(* IEC 61131-3 sources: std_i2980_v2.06_cp053/Source/IMM/ieccontrol/ExceptionInterpretation1 (part 2) *)

(* ---- FBODCErrorHandler.pu ---- *)
IMPORT_OVER_LISTFILE
 tyAlarmParams
, tySubID

END_IMPORT

FUNCTION_BLOCK FBODCErrorHandler #DUMMY_EDIT_BLOCK

VAR_INPUT
 iErrorKind : INT;
 iComponentNr : DINT;
 iErrorNr : DINT;
 AlarmParameters : tyAlarmParams;
END_VAR

VAR_IN_OUT
 SubID : tySubID;
END_VAR

VAR_OUTPUT
 bOpenWatchdog : BOOL;
 bSetAlarm : BOOL;
 AlarmID : ALARM;
 sParam1 : STRING(255);
 sParam2 : STRING(255);
END_VAR

SYSTEM_OBJECT
 erODCBuilderGeneralError : ALARM;
 erODCBuilderNoSignature : ALARM;
 erODCBuilderFileformat : ALARM;
 erODCBuilderInvalidSignature : ALARM;
 erODCBuilderInsertPosNotAvail : ALARM;
 erODCBuilderInsertBefNotAllow : ALARM;
 erODCBuilderInsertAfterNotAllow : ALARM;
 erODCBuilderMoveNotAvailable : ALARM;
 erODCBuilderError : ALARM;
 erODCBuilderSyntaxError : ALARM;
 erODCBuilderWarning : ALARM;
 erODCBuilderWarningFile : ALARM;
 erODCBuilderMultipleBaseSequ : ALARM;
 erODCBuilderPriorityCollision : ALARM;
 erODCBuilderBaseSeqNotFound : ALARM;
 erODCBuilderInstancePriority : ALARM;
 erODCBuilderParserException : ALARM;
 erODCCouldNotCreateLogFile : ALARM;
 erODCBuilderFirstMovement : ALARM;
 erODCBuilderLastMovement : ALARM;
 erODCBuilderSelectorVarValue : ALARM;
 erODCBuilderIllegalDominantMove : ALARM;
 erODCBuilderInsertParallel : ALARM;
 erODCBuilderInvalidCreateSequ : ALARM;
 erODCBuilderElementAlreadyUsed : ALARM;
 erODCBuilderArrayTooSmall : ALARM;
 erODCBuilderInternalError : ALARM;
 erODCMLFExpireTime : ALARM;
END_OBJECT

VAR
 ErrorCounter : DINT (* for making sure errors get a unique numer *);
END_VAR
#BEGIN_EDIT_BLOCK
(**************************************** WARNING ********************************************
 *** The KEBA Kemro K2 System including software is not intended for safety control tasks! ***
 ***                       For further information see Comment tab!                        ***
 *********************************************************************************************)

(* ERROR *********************************************************************************)
IF (iErrorKind = cErrorKind_Error) THEN
   CASE iComponentNr OF
      6750:   //ODC
         bSetAlarm := TRUE;
         bOpenWatchdog := FALSE;
         SubID[3] := ErrorCounter;

         CASE iErrorNr OF
            1: (* "BaseSequenceFile does not exist in %1" *)
               AlarmID := erODCBuilderBaseSeqNotFound;
               sParam1 := AlarmParameters[1];

            2: (* "ODCBuilder Parser Syntax Error: %1 - file %2 line %3 col %4" *)
               AlarmID := erODCBuilderSyntaxError;
               sParam1 := AlarmParameters[1];
               sParam2 := AlarmParameters[2];
               SubID[3] := STRING_TO_DINT(AlarmParameters[3]);
               SubID[4] := STRING_TO_DINT(AlarmParameters[4]);

            3: (* "ODCBuilder Parser Error: %1 - file %2 line %3 col %4" *)
               AlarmID := erODCBuilderError;
               sParam1 := AlarmParameters[1];
               sParam2 := AlarmParameters[2];
               SubID[3] := STRING_TO_DINT(AlarmParameters[3]);
               SubID[4] := STRING_TO_DINT(AlarmParameters[4]);

            (* 4, 5: WARNING *)

            6: (* "ODCBuilder Parser Exception: %1" *)
               AlarmID := erODCBuilderParserException;
               sParam1 := AlarmParameters[1];
               bOpenWatchdog := TRUE;

            (* 100: WARNING *)

            101: (* "ODCBuilder: fileformat version %1 of file %2 not supported" *)
               AlarmID := erODCBuilderFileformat;
               sParam1 := CONCAT(AlarmParameters[1], '.', AlarmParameters[2]);
               sParam2 := AlarmParameters[3];

            102: (* "ODCBuilder: first movement in base sequence must be ODC.BeginSequence" *)
               AlarmID := erODCBuilderFirstMovement;

            103: (* "ODCBuilder: last movement in base sequence must be ODC.EndSequence" *)
               AlarmID := erODCBuilderLastMovement;

            (* 104 WARNING *)

            105: (* "ODCBuilder: File %1 has an invalid signature" *)
               AlarmID := erODCBuilderInvalidSignature;
               sParam1 := AlarmParameters[1];

            106: (* "ODCBuilder: BaseSequence is already defined - file %1" *)
               AlarmID := erODCBuilderMultipleBaseSequ;
               //alarm should only be displayed once, no matter how many base sequences are found
               SubID[3] := 0;

            110: (* "ODCBuilder: cannot get value for selector variable %1 in file %2" *)
               //check type of selector variable (for example REAL variables are not allowed)
               AlarmID := erODCBuilderSelectorVarValue;
               sParam1 := AlarmParameters[1];
               sParam2 := AlarmParameters[2];

            112: (* "ODCBuilder: movement %1 not available in movementlist" *)
               // movement to insert not found in sv_ODCMovements
               // sMoveId of the sv_MoveXxx is not set or it is different from the identifier used in the text file
               AlarmID := erODCBuilderMoveNotAvailable;
               sParam1 := AlarmParameters[1];
               sParam2 := AlarmParameters[2];

            113: (* "ODCBuilder: illegal dominant movement %1 in insert block %2" *)
               AlarmID := erODCBuilderIllegalDominantMove;
               sParam1 := AlarmParameters[1];
               sParam2 := CONCAT(AlarmParameters[2], ' ', AlarmParameters[3], '=', AlarmParameters[4]);

            114: (* "ODCBuilder: instance priority for movement %1 insert block %2 necessary" *)
               // several insert statements or instances of the same device try to insert at the same position with the same priority
               // Use ODC->Priority Check in Notepad++ to check for priority conflicts
               // Change the priority of the conflicting insert statement
               // Or in case there are several instances(eg. Core, AirValve, ...) add a instance priority (pInstancePrio^ in sv_MoveXxx)
               AlarmID := erODCBuilderInstancePriority;
               sParam1 := AlarmParameters[1];
               sParam2 := CONCAT(AlarmParameters[2], ' ', AlarmParameters[3], '=', AlarmParameters[4]);

            115: (* "ODCBuilder: same insert and instance priority for 2 movements (priority collision)" *)
               AlarmID := erODCBuilderPriorityCollision;
               sParam1 := AlarmParameters[1];
               sParam2 := AlarmParameters[2];

            120: (* "ODCBuilder: insert position %1 for insert block %2 not found in sequence" *)
               // when %1 is not in base sequence but another file, most likely cause is a wrong priority.
               // %1 is not inserted yet when somebody else tries to use it as a insert position
               AlarmID := erODCBuilderInsertPosNotAvail;
               sParam1 := AlarmParameters[1];
               sParam2 := CONCAT(AlarmParameters[2], ' ', AlarmParameters[3], '=', AlarmParameters[4]);

            121: (* "ODCBuilder: insert of insert block %1 before ODC.BeginSequence not allowed" *)
               AlarmID := erODCBuilderInsertBefNotAllow;
               sParam1 := CONCAT(AlarmParameters[2], ' ', AlarmParameters[3], '=', AlarmParameters[4]);

            123: (* "ODCBuilder: insert of insert block %1 after ODC.EndSequence not allowed" *)
               AlarmID := erODCBuilderInsertAfterNotAllow;
               sParam1 := CONCAT(AlarmParameters[2], ' ', AlarmParameters[3], '=', AlarmParameters[4]);

            124: (* "ODCBuilder: invalid insert parallel at %1 of insert block %2" *)
               AlarmID := erODCBuilderInsertParallel;
               sParam1 := AlarmParameters[1];
               sParam2 := CONCAT(AlarmParameters[2], ' ', AlarmParameters[3], '=', AlarmParameters[4]);

            125: (* "ODCBuilder: sequence array (height %1 width %2) is to small (line %3 column %4)" *)
               AlarmID := erODCBuilderArrayTooSmall;
               SubID[1] := STRING_TO_DINT(AlarmParameters[1]);
               SubID[2] := STRING_TO_DINT(AlarmParameters[2]);
               SubID[3] := STRING_TO_DINT(AlarmParameters[3]);
               SubID[4] := STRING_TO_DINT(AlarmParameters[4]);

            126: (* "ODCBuilder: invalid call of CreateSequence - init error %1 occured" *)
               AlarmID := erODCBuilderInvalidCreateSequ;
               sParam1 := AlarmParameters[1];

            127: (* "ODCBuilder: invalid call of CreateSequence - init error %1 occured" *)
               AlarmID := erODCBuilderElementAlreadyUsed;
               sParam1 := AlarmParameters[1];
               sParam2 := AlarmParameters[2];

            199: (* "ODCBuilder: internal error: %1" *)
               AlarmID := erODCBuilderInternalError;
               sParam1 := AlarmParameters[1];

            1000: (* "MLF: Firmware detected exceeding expire time" *)
               AlarmID := erODCMLFExpireTime;

         ELSE (* any other alarm *)
            AlarmID := erODCBuilderGeneralError;
            bOpenWatchdog := TRUE;

         END_CASE;
   END_CASE;
   (* WARNING *****************************************************************************)
ELSIF (iErrorKind = cErrorKind_Warning) THEN
   bOpenWatchdog := FALSE;
   bSetAlarm := TRUE;

   CASE iComponentNr OF
      6750:   //ODC
         CASE iErrorNr OF
            4: (* "ODCBuilder Parser Warning: %1 - file %2 line %3 col %4" *)
               AlarmID := erODCBuilderWarningFile;
               sParam1 := AlarmParameters[1];
               sParam2 := AlarmParameters[2];
               SubID[3] := STRING_TO_DINT(AlarmParameters[3]);
               SubID[4] := STRING_TO_DINT(AlarmParameters[4]);

            5: (* "ODCBuilder Parser Warning: %1" *)
               AlarmID := erODCBuilderWarning;
               sParam1 := AlarmParameters[1];
               SubID[3] := ErrorCounter;

            100: (* "ODCBuilder cannot create logfile %1" *)
               AlarmID := erODCCouldNotCreateLogFile;
               sParam1 := AlarmParameters[1];

            104: (* "ODCBuilder: File %1 has no signature" *)
               AlarmID := erODCBuilderNoSignature;
               sParam1 := AlarmParameters[1];
               SubID[3] := ErrorCounter;
         END_CASE;
   END_CASE;
END_IF;
ErrorCounter := ErrorCounter + 1;

;#END_EDIT_BLOCK END_FUNCTION_BLOCK

#END_OF_IEC_PART

@Puma @IecEditor 6 97 @Pou 25
@@@BEG_Comment@@@

@@@END_Comment@@@

@BEG_Contents

@BEG_Func
@RT(17)FuncTreeContainer
0
@END_Func

@BEG_Const
@RT(18)ConstTreeContainer
0
@END_Const

@BEG_Export

@BEG_Kind
@FUNCTION_BLOCK @RT(17)FBODCErrorHandler @STRUCTURED_TEXT
@RT(0) @RT(0) @RT(0)
@END_Kind

@BEG_Dcl
@RT(16)DclTreeContainer
39
@Var @RT(10)iErrorKind @RT(0) @T @F @DT @RT(3)INT @RT(0) @T @T @BASIC 0 @F
@F @F
@T
@BEG_Attrib
3 @RT(0) @RT(0) @RT(0)
@END_Attrib
1 1 @F @F @F @F

@Var @RT(12)iComponentNr @RT(0) @T @F @DT @RT(4)DINT @RT(0) @T @T @BASIC 0 @F
@F @F
@T
@BEG_Attrib
3 @RT(0) @RT(0) @RT(0)
@END_Attrib
1 1 @F @F @F @F

@Var @RT(8)iErrorNr @RT(0) @T @F @DT @RT(4)DINT @RT(0) @T @T @BASIC 0 @F
@F @F
@T
@BEG_Attrib
3 @RT(0) @RT(0) @RT(0)
@END_Attrib
1 1 @F @F @F @F

@Var @RT(15)AlarmParameters @RT(0) @T @T @DERIVED 0 @T @T @DT @RT(13)tyAlarmParams @RT(0) @T @T @UNKNOWN 0 @F
@F @F
@T
@BEG_Attrib
3 @RT(0) @RT(0) @RT(0)
@END_Attrib
1 1 @F @F @F @F

@Var @RT(5)SubID @RT(0) @T @T @DERIVED 0 @F @RT(7)tySubID @F
@T
@BEG_Attrib
3 @RT(0) @RT(0) @RT(0)
@END_Attrib
1 2 @F @F @F @F

@Var @RT(13)bOpenWatchdog @RT(0) @T @F @DT @RT(4)BOOL @RT(0) @T @T @BASIC 0 @F
@F @F
@T
@BEG_Attrib
3 @RT(0) @RT(0) @RT(0)
@END_Attrib
1 3 @F @F @F @F

@Var @RT(9)bSetAlarm @RT(0) @T @F @DT @RT(4)BOOL @RT(0) @T @T @BASIC 0 @F
@F @F
@T
@BEG_Attrib
3 @RT(0) @RT(0) @RT(0)
@END_Attrib
1 3 @F @F @F @F

@Var @RT(7)AlarmID @RT(0) @T @F @DT @RT(5)ALARM @RT(0) @T @T @BASIC 0 @F
@F @F
@T
@BEG_Attrib
3 @RT(0) @RT(0) @RT(0)
@END_Attrib
1 3 @F @F @F @F

@Var @RT(7)sParam1 @RT(0) @T @F @DT @RT(11)STRING(255) @RT(0) @T @T @STRING 0 @F @RT(3)255 @F
@F @F
@T
@BEG_Attrib
3 @RT(0) @RT(0) @RT(0)
@END_Attrib
1 3 @F @F @F @F

@Var @RT(7)sParam2 @RT(0) @T @F @DT @RT(11)STRING(255) @RT(0) @T @T @STRING 0 @F @RT(3)255 @F
@F @F
@T
@BEG_Attrib
3 @RT(0) @RT(0) @RT(0)
@END_Attrib
1 3 @F @F @F @F

@Var @RT(24)erODCBuilderGeneralError @RT(0) @T @T @RENAMED 0 @T @T @DT @RT(5)ALARM @RT(0) @T @T @BASIC 0 @F
@F @F
@T
@BEG_Attrib
3 @RT(0) @RT(0) @RT(0)
@END_Attrib
1 7 @F @F @F @F

@Var @RT(23)erODCBuilderNoSignature @RT(0) @T @F @DT @RT(5)ALARM @RT(0) @T @T @BASIC 0 @F
@F @F
@T
@BEG_Attrib
3 @RT(0) @RT(0) @RT(0)
@END_Attrib
1 7 @F @F @F @F

@Var @RT(22)erODCBuilderFileformat @RT(0) @T @F @DT @RT(5)ALARM @RT(0) @T @T @BASIC 0 @F
@F @F
@T
@BEG_Attrib
3 @RT(0) @RT(0) @RT(0)
@END_Attrib
1 7 @F @F @F @F

@Var @RT(28)erODCBuilderInvalidSignature @RT(0) @T @F @DT @RT(5)ALARM @RT(0) @T @T @BASIC 0 @F
@F @F
@T
@BEG_Attrib
3 @RT(0) @RT(0) @RT(0)
@END_Attrib
1 7 @F @F @F @F

@Var @RT(29)erODCBuilderInsertPosNotAvail @RT(0) @T @F @DT @RT(5)ALARM @RT(0) @T @T @BASIC 0 @F
@F @F
@T
@BEG_Attrib
3 @RT(0) @RT(0) @RT(0)
@END_Attrib
1 7 @F @F @F @F

@Var @RT(29)erODCBuilderInsertBefNotAllow @RT(0) @T @F @DT @RT(5)ALARM @RT(0) @T @T @BASIC 0 @F
@F @F
@T
@BEG_Attrib
3 @RT(0) @RT(0) @RT(0)
@END_Attrib
1 7 @F @F @F @F

@Var @RT(31)erODCBuilderInsertAfterNotAllow @RT(0) @T @F @DT @RT(5)ALARM @RT(0) @T @T @BASIC 0 @F
@F @F
@T
@BEG_Attrib
3 @RT(0) @RT(0) @RT(0)
@END_Attrib
1 7 @F @F @F @F

@Var @RT(28)erODCBuilderMoveNotAvailable @RT(0) @T @F @DT @RT(5)ALARM @RT(0) @T @T @BASIC 0 @F
@F @F
@T
@BEG_Attrib
3 @RT(0) @RT(0) @RT(0)
@END_Attrib
1 7 @F @F @F @F

@Var @RT(17)erODCBuilderError @RT(0) @T @F @DT @RT(5)ALARM @RT(0) @T @T @BASIC 0 @F
@F @F
@T
@BEG_Attrib
3 @RT(0) @RT(0) @RT(0)
@END_Attrib
1 7 @F @F @F @F

@Var @RT(23)erODCBuilderSyntaxError @RT(0) @T @F @DT @RT(5)ALARM @RT(0) @T @T @BASIC 0 @F
@F @F
@T
@BEG_Attrib
3 @RT(0) @RT(0) @RT(0)
@END_Attrib
1 7 @F @F @F @F

@Var @RT(19)erODCBuilderWarning @RT(0) @T @F @DT @RT(5)ALARM @RT(0) @T @T @BASIC 0 @F
@F @F
@T
@BEG_Attrib
3 @RT(0) @RT(0) @RT(0)
@END_Attrib
1 7 @F @F @F @F

@Var @RT(23)erODCBuilderWarningFile @RT(0) @T @F @DT @RT(5)ALARM @RT(0) @T @T @BASIC 0 @F
@F @F
@T
@BEG_Attrib
3 @RT(0) @RT(0) @RT(0)
@END_Attrib
1 7 @F @F @F @F

@Var @RT(28)erODCBuilderMultipleBaseSequ @RT(0) @T @F @DT @RT(5)ALARM @RT(0) @T @T @BASIC 0 @F
@F @F
@T
@BEG_Attrib
3 @RT(0) @RT(0) @RT(0)
@END_Attrib
1 7 @F @F @F @F

@Var @RT(29)erODCBuilderPriorityCollision @RT(0) @T @F @DT @RT(5)ALARM @RT(0) @T @T @BASIC 0 @F
@F @F
@T
@BEG_Attrib
3 @RT(0) @RT(0) @RT(0)
@END_Attrib
1 7 @F @F @F @F

@Var @RT(27)erODCBuilderBaseSeqNotFound @RT(0) @T @T @RENAMED 0 @T @T @DT @RT(5)ALARM @RT(0) @T @T @BASIC 0 @F
@F @F
@T
@BEG_Attrib
3 @RT(0) @RT(0) @RT(0)
@END_Attrib
1 7 @F @F @F @F

@Var @RT(28)erODCBuilderInstancePriority @RT(0) @T @T @RENAMED 0 @T @T @DT @RT(5)ALARM @RT(0) @T @T @BASIC 0 @F
@F @F
@T
@BEG_Attrib
3 @RT(0) @RT(0) @RT(0)
@END_Attrib
1 7 @F @F @F @F

@Var @RT(12)ErrorCounter @RT(0) @T @F @DT @RT(4)DINT @RT(0) @T @T @BASIC 0 @F
@F @F
@T
@BEG_Attrib
3 @RT(0) @RT(41)for making sure errors get a unique numer @RT(0)
@END_Attrib
1 0 @F @F @F @F

@Var @RT(27)erODCBuilderParserException @RT(0) @T @F @DT @RT(5)ALARM @RT(0) @T @T @BASIC 0 @F
@F @F
@T
@BEG_Attrib
3 @RT(0) @RT(0) @RT(0)
@END_Attrib
1 7 @F @F @F @F

@Var @RT(26)erODCCouldNotCreateLogFile @RT(0) @T @F @DT @RT(5)ALARM @RT(0) @T @T @BASIC 0 @F
@F @F
@T
@BEG_Attrib
3 @RT(0) @RT(0) @RT(0)
@END_Attrib
1 7 @F @F @F @F

@Var @RT(25)erODCBuilderFirstMovement @RT(0) @T @F @DT @RT(5)ALARM @RT(0) @T @T @BASIC 0 @F
@F @F
@T
@BEG_Attrib
3 @RT(0) @RT(0) @RT(0)
@END_Attrib
1 7 @F @F @F @F

@Var @RT(24)erODCBuilderLastMovement @RT(0) @T @F @DT @RT(5)ALARM @RT(0) @T @T @BASIC 0 @F
@F @F
@T
@BEG_Attrib
3 @RT(0) @RT(0) @RT(0)
@END_Attrib
1 7 @F @F @F @F

@Var @RT(28)erODCBuilderSelectorVarValue @RT(0) @T @F @DT @RT(5)ALARM @RT(0) @T @T @BASIC 0 @F
@F @F
@T
@BEG_Attrib
3 @RT(0) @RT(0) @RT(0)
@END_Attrib
1 7 @F @F @F @F

@Var @RT(31)erODCBuilderIllegalDominantMove @RT(0) @T @F @DT @RT(5)ALARM @RT(0) @T @T @BASIC 0 @F
@F @F
@T
@BEG_Attrib
3 @RT(0) @RT(0) @RT(0)
@END_Attrib
1 7 @F @F @F @F

@Var @RT(26)erODCBuilderInsertParallel @RT(0) @T @F @DT @RT(5)ALARM @RT(0) @T @T @BASIC 0 @F
@F @F
@T
@BEG_Attrib
3 @RT(0) @RT(0) @RT(0)
@END_Attrib
1 7 @F @F @F @F

@Var @RT(29)erODCBuilderInvalidCreateSequ @RT(0) @T @F @DT @RT(5)ALARM @RT(0) @T @T @BASIC 0 @F
@F @F
@T
@BEG_Attrib
3 @RT(0) @RT(0) @RT(0)
@END_Attrib
1 7 @F @F @F @F

@Var @RT(30)erODCBuilderElementAlreadyUsed @RT(0) @T @F @DT @RT(5)ALARM @RT(0) @T @T @BASIC 0 @F
@F @F
@T
@BEG_Attrib
3 @RT(0) @RT(0) @RT(0)
@END_Attrib
1 7 @F @F @F @F

@Var @RT(25)erODCBuilderArrayTooSmall @RT(0) @T @F @DT @RT(5)ALARM @RT(0) @T @T @BASIC 0 @F
@F @F
@T
@BEG_Attrib
3 @RT(0) @RT(0) @RT(0)
@END_Attrib
1 7 @F @F @F @F

@Var @RT(25)erODCBuilderInternalError @RT(0) @T @F @DT @RT(5)ALARM @RT(0) @T @T @BASIC 0 @F
@F @F
@T
@BEG_Attrib
3 @RT(0) @RT(0) @RT(0)
@END_Attrib
1 7 @F @F @F @F

@Var @RT(18)erODCMLFExpireTime @RT(0) @T @T @RENAMED 0 @T @T @DT @RT(5)ALARM @RT(0) @T @T @BASIC 0 @F
@F @F
@T
@BEG_Attrib
3 @RT(0) @RT(0) @RT(0)
@END_Attrib
1 7 @F @F @F @F

@END_Dcl

@END_Export

@BEG_Body
@TL(177)
(**************************************** WARNING ********************************************
 *** The KEBA Kemro K2 System including software is not intended for safety control tasks! ***
 ***                       For further information see Comment tab!                        ***
 *********************************************************************************************)

(* ERROR *********************************************************************************)
IF (iErrorKind = cErrorKind_Error) THEN
   CASE iComponentNr OF
      6750:   //ODC
         bSetAlarm := TRUE;
         bOpenWatchdog := FALSE;
         SubID[3] := ErrorCounter;

         CASE iErrorNr OF
            1: (* "BaseSequenceFile does not exist in %1" *)
               AlarmID := erODCBuilderBaseSeqNotFound;
               sParam1 := AlarmParameters[1];

            2: (* "ODCBuilder Parser Syntax Error: %1 - file %2 line %3 col %4" *)
               AlarmID := erODCBuilderSyntaxError;
               sParam1 := AlarmParameters[1];
               sParam2 := AlarmParameters[2];
               SubID[3] := STRING_TO_DINT(AlarmParameters[3]);
               SubID[4] := STRING_TO_DINT(AlarmParameters[4]);

            3: (* "ODCBuilder Parser Error: %1 - file %2 line %3 col %4" *)
               AlarmID := erODCBuilderError;
               sParam1 := AlarmParameters[1];
               sParam2 := AlarmParameters[2];
               SubID[3] := STRING_TO_DINT(AlarmParameters[3]);
               SubID[4] := STRING_TO_DINT(AlarmParameters[4]);

            (* 4, 5: WARNING *)

            6: (* "ODCBuilder Parser Exception: %1" *)
               AlarmID := erODCBuilderParserException;
               sParam1 := AlarmParameters[1];
               bOpenWatchdog := TRUE;

            (* 100: WARNING *)

            101: (* "ODCBuilder: fileformat version %1 of file %2 not supported" *)
               AlarmID := erODCBuilderFileformat;
               sParam1 := CONCAT(AlarmParameters[1], '.', AlarmParameters[2]);
               sParam2 := AlarmParameters[3];

            102: (* "ODCBuilder: first movement in base sequence must be ODC.BeginSequence" *)
               AlarmID := erODCBuilderFirstMovement;

            103: (* "ODCBuilder: last movement in base sequence must be ODC.EndSequence" *)
               AlarmID := erODCBuilderLastMovement;

            (* 104 WARNING *)

            105: (* "ODCBuilder: File %1 has an invalid signature" *)
               AlarmID := erODCBuilderInvalidSignature;
               sParam1 := AlarmParameters[1];

            106: (* "ODCBuilder: BaseSequence is already defined - file %1" *)
               AlarmID := erODCBuilderMultipleBaseSequ;
               //alarm should only be displayed once, no matter how many base sequences are found
               SubID[3] := 0;

            110: (* "ODCBuilder: cannot get value for selector variable %1 in file %2" *)
               //check type of selector variable (for example REAL variables are not allowed)
               AlarmID := erODCBuilderSelectorVarValue;
               sParam1 := AlarmParameters[1];
               sParam2 := AlarmParameters[2];

            112: (* "ODCBuilder: movement %1 not available in movementlist" *)
               // movement to insert not found in sv_ODCMovements
               // sMoveId of the sv_MoveXxx is not set or it is different from the identifier used in the text file
               AlarmID := erODCBuilderMoveNotAvailable;
               sParam1 := AlarmParameters[1];
               sParam2 := AlarmParameters[2];

            113: (* "ODCBuilder: illegal dominant movement %1 in insert block %2" *)
               AlarmID := erODCBuilderIllegalDominantMove;
               sParam1 := AlarmParameters[1];
               sParam2 := CONCAT(AlarmParameters[2], ' ', AlarmParameters[3], '=', AlarmParameters[4]);

            114: (* "ODCBuilder: instance priority for movement %1 insert block %2 necessary" *)
               // several insert statements or instances of the same device try to insert at the same position with the same priority
               // Use ODC->Priority Check in Notepad++ to check for priority conflicts
               // Change the priority of the conflicting insert statement
               // Or in case there are several instances(eg. Core, AirValve, ...) add a instance priority (pInstancePrio^ in sv_MoveXxx)
               AlarmID := erODCBuilderInstancePriority;
               sParam1 := AlarmParameters[1];
               sParam2 := CONCAT(AlarmParameters[2], ' ', AlarmParameters[3], '=', AlarmParameters[4]);

            115: (* "ODCBuilder: same insert and instance priority for 2 movements (priority collision)" *)
               AlarmID := erODCBuilderPriorityCollision;
               sParam1 := AlarmParameters[1];
               sParam2 := AlarmParameters[2];

            120: (* "ODCBuilder: insert position %1 for insert block %2 not found in sequence" *)
               // when %1 is not in base sequence but another file, most likely cause is a wrong priority.
               // %1 is not inserted yet when somebody else tries to use it as a insert position
               AlarmID := erODCBuilderInsertPosNotAvail;
               sParam1 := AlarmParameters[1];
               sParam2 := CONCAT(AlarmParameters[2], ' ', AlarmParameters[3], '=', AlarmParameters[4]);

            121: (* "ODCBuilder: insert of insert block %1 before ODC.BeginSequence not allowed" *)
               AlarmID := erODCBuilderInsertBefNotAllow;
               sParam1 := CONCAT(AlarmParameters[2], ' ', AlarmParameters[3], '=', AlarmParameters[4]);

            123: (* "ODCBuilder: insert of insert block %1 after ODC.EndSequence not allowed" *)
               AlarmID := erODCBuilderInsertAfterNotAllow;
               sParam1 := CONCAT(AlarmParameters[2], ' ', AlarmParameters[3], '=', AlarmParameters[4]);

            124: (* "ODCBuilder: invalid insert parallel at %1 of insert block %2" *)
               AlarmID := erODCBuilderInsertParallel;
               sParam1 := AlarmParameters[1];
               sParam2 := CONCAT(AlarmParameters[2], ' ', AlarmParameters[3], '=', AlarmParameters[4]);

            125: (* "ODCBuilder: sequence array (height %1 width %2) is to small (line %3 column %4)" *)
               AlarmID := erODCBuilderArrayTooSmall;
               SubID[1] := STRING_TO_DINT(AlarmParameters[1]);
               SubID[2] := STRING_TO_DINT(AlarmParameters[2]);
               SubID[3] := STRING_TO_DINT(AlarmParameters[3]);
               SubID[4] := STRING_TO_DINT(AlarmParameters[4]);

            126: (* "ODCBuilder: invalid call of CreateSequence - init error %1 occured" *)
               AlarmID := erODCBuilderInvalidCreateSequ;
               sParam1 := AlarmParameters[1];

            127: (* "ODCBuilder: invalid call of CreateSequence - init error %1 occured" *)
               AlarmID := erODCBuilderElementAlreadyUsed;
               sParam1 := AlarmParameters[1];
               sParam2 := AlarmParameters[2];

            199: (* "ODCBuilder: internal error: %1" *)
               AlarmID := erODCBuilderInternalError;
               sParam1 := AlarmParameters[1];

            1000: (* "MLF: Firmware detected exceeding expire time" *)
               AlarmID := erODCMLFExpireTime;

         ELSE (* any other alarm *)
            AlarmID := erODCBuilderGeneralError;
            bOpenWatchdog := TRUE;

         END_CASE;
   END_CASE;
   (* WARNING *****************************************************************************)
ELSIF (iErrorKind = cErrorKind_Warning) THEN
   bOpenWatchdog := FALSE;
   bSetAlarm := TRUE;

   CASE iComponentNr OF
      6750:   //ODC
         CASE iErrorNr OF
            4: (* "ODCBuilder Parser Warning: %1 - file %2 line %3 col %4" *)
               AlarmID := erODCBuilderWarningFile;
               sParam1 := AlarmParameters[1];
               sParam2 := AlarmParameters[2];
               SubID[3] := STRING_TO_DINT(AlarmParameters[3]);
               SubID[4] := STRING_TO_DINT(AlarmParameters[4]);

            5: (* "ODCBuilder Parser Warning: %1" *)
               AlarmID := erODCBuilderWarning;
               sParam1 := AlarmParameters[1];
               SubID[3] := ErrorCounter;

            100: (* "ODCBuilder cannot create logfile %1" *)
               AlarmID := erODCCouldNotCreateLogFile;
               sParam1 := AlarmParameters[1];

            104: (* "ODCBuilder: File %1 has no signature" *)
               AlarmID := erODCBuilderNoSignature;
               sParam1 := AlarmParameters[1];
               SubID[3] := ErrorCounter;
         END_CASE;
   END_CASE;
END_IF;
ErrorCounter := ErrorCounter + 1;

@END_Body

@END_Contents

(* ---- ABCPUTemperature.pu ---- *)
(*
@h    ! WARNING !
@h    The Kemro K2 system (including software) only meets category B according to EN 954-1,
@h    thus it is not intended for usage in safety-relevant control applications in the field
@h    of personal safety (e.g. emergency stop).
@h    To implement potentially necessary safety-relevant control tasks, always use additional
@h    external safety devices that are intended for the particular purpose, and meet the necessary
@h    functional safety.
@h    For further information see EN 954-1 (EN ISO 13849-1) and/or the K2-x00 user manual, chapter
@h    "CE conformity, directives and standards".

polling of CPU Temperature
-> can be started and stopped
-> Alarm to finish cycle and stop if temperature limit is reached
-> temperature limit depends on cpu

@FunctionID: CR_0034081

*)

IMPORT_OVER_LISTFILE
 GET_TEMP
, SET_ALARM
, RESET_ALARM
, KCAT_HandleData
, KCAT_Status
, KSYS_TempId
, KSYS_GetTemp_Data

END_IMPORT

ALGORITHM_BLOCK ABCPUTemperature #DUMMY_EDIT_BLOCK

SYSTEM_OBJECT
 TaskSlow : TASK;
 erCPUTempHigh : ALARM;
END_OBJECT

VAR
 mbInit : BOOL;
 mbStart : BOOL;
 mrTemperatureLimit : REAL;
END_VAR

ALGORITHM aStart

#BEGIN_EDIT_BLOCK
(**************************************** WARNING ********************************************
 *** The KEBA Kemro K2 System including software is not intended for safety control tasks! ***
 ***                       For further information see Comment tab!                        ***
 *********************************************************************************************)

mbStart := TRUE;
START_PROCESS_ALGORITHM(paRun)

;#END_EDIT_BLOCK END_ALGORITHM

ALGORITHM aStop

#BEGIN_EDIT_BLOCK
(**************************************** WARNING ********************************************
 *** The KEBA Kemro K2 System including software is not intended for safety control tasks! ***
 ***                       For further information see Comment tab!                        ***
 *********************************************************************************************)

mbStart := FALSE;

;#END_EDIT_BLOCK END_ALGORITHM

PROCESS_ALGORITHM paInit ON TaskSlow AUTOSTART

VAR
 hdl : KCAT_HandleData;
 sPlatform : STRING(10);
 state : KCAT_Status;
 dummy : DINT;
END_VAR
#BEGIN_EDIT_BLOCK
(**************************************** WARNING ********************************************
 *** The KEBA Kemro K2 System including software is not intended for safety control tasks! ***
 ***                       For further information see Comment tab!                        ***
 *********************************************************************************************)

//get hardware platform
hdl := KCAT_GetHandle('IRT.Platform');
IF hdl.Status = KCAT_Status_OK THEN
   state := KCAT_GetValue(Handle := hdl.Handle, Buffer := sPlatform);
END_IF;

IF sPlatform = 'PPC' THEN
   mrTemperatureLimit := 83.0; //PPC
ELSIF sPlatform = 'x86' THEN
   mrTemperatureLimit := 115.0; //Intel
ELSE
   //unknown platform -> set trace and use lower temperature limit
   dummy := Print('!!! ABCPUTemperature - paInit: could not detect hardware platform !!!');
   mrTemperatureLimit := 83.0;
END_IF;

mbInit := TRUE;
STOP_PROCESS_ALGORITHM();

;#END_EDIT_BLOCK END_ALGORITHM

PROCESS_ALGORITHM paRun ON TaskSlow

VAR
 TempID : KSYS_TempId := KSYS_TempID_MAB;
 TempData : KSYS_GetTemp_Data;
 iCycleRed : DINT;
 bAlarmSet : BOOL;
END_VAR
#BEGIN_EDIT_BLOCK
(**************************************** WARNING ********************************************
 *** The KEBA Kemro K2 System including software is not intended for safety control tasks! ***
 ***                       For further information see Comment tab!                        ***
 *********************************************************************************************)
IF (NOT mbStart) THEN
    iCycleRed := 0;
    STOP_PROCESS_ALGORITHM();
    RETURN;
END_IF;

IF (NOT mbInit) THEN
    RETURN;
END_IF;

IF ((iCycleRed MOD 64) = 0) THEN // about every 0,5 min
  TempData := GET_TEMP(TempID);

  IF (TempData.Temp >= REAL_TO_DINT(mrTemperatureLimit)) THEN
        SET_ALARM(Name := erCPUTempHigh, Param1 := DINT_TO_STRING(TempData.Temp));
        bAlarmSet := TRUE;
  END_IF;

  IF (TempData.Temp < (REAL_TO_DINT(mrTemperatureLimit) - 1)) THEN
        IF bAlarmSet THEN
            RESET_ALARM(Name := erCPUTempHigh);
            bAlarmSet := FALSE;
        END_IF;
  END_IF;

END_IF;

iCycleRed := iCycleRed + 1;

;#END_EDIT_BLOCK END_ALGORITHM

END_ALGORITHM_BLOCK

#END_OF_IEC_PART

@Puma @IecEditor 6 80 @Pou 25
@@@BEG_Comment@@@
@h    ! WARNING !
@h    The Kemro K2 system (including software) only meets category B according to EN 954-1,
@h    thus it is not intended for usage in safety-relevant control applications in the field
@h    of personal safety (e.g. emergency stop).
@h    To implement potentially necessary safety-relevant control tasks, always use additional
@h    external safety devices that are intended for the particular purpose, and meet the necessary
@h    functional safety.
@h    For further information see EN 954-1 (EN ISO 13849-1) and/or the K2-x00 user manual, chapter
@h    "CE conformity, directives and standards".

polling of CPU Temperature
-> can be started and stopped
-> Alarm to finish cycle and stop if temperature limit is reached
-> temperature limit depends on cpu

@FunctionID: CR_0034081

@@@END_Comment@@@

@BEG_Contents

@BEG_Func
@RT(17)FuncTreeContainer
3
@Var @RT(8)GET_TEMP @RT(0) @T @T @DERIVED 0 @F @RT(22)KEBA_STANDARD_FUNCTION @F
@T
@BEG_Attrib
0 @RT(0) @RT(0)
@END_Attrib
1 1 @F @F @F @F

@Var @RT(9)SET_ALARM @RT(0) @T @T @DERIVED 0 @F @RT(23)KEBA_STANDARD_PROCEDURE @F
@T
@BEG_Attrib
0 @RT(0) @RT(0)
@END_Attrib
1 1 @F @F @F @F

@Var @RT(11)RESET_ALARM @RT(0) @T @T @DERIVED 0 @F @RT(23)KEBA_STANDARD_PROCEDURE @F
@T
@BEG_Attrib
0 @RT(0) @RT(0)
@END_Attrib
1 1 @F @F @F @F

@END_Func

@BEG_Const
@RT(18)ConstTreeContainer
0
@END_Const

@BEG_Export

@BEG_Kind
@ALGORITHM_BLOCK @RT(16)ABCPUTemperature @STRUCTURED_TEXT
@RT(0) @RT(0) @RT(0)
@END_Kind

@BEG_Dcl
@RT(16)DclTreeContainer
5
@Var @RT(6)mbInit @RT(0) @T @F @DT @RT(4)BOOL @RT(0) @T @T @BASIC 0 @F
@F @F
@T
@BEG_Attrib
3 @RT(0) @RT(0) @RT(0)
@END_Attrib
1 0 @F @F @F @F

@Var @RT(7)mbStart @RT(0) @T @F @DT @RT(4)BOOL @RT(0) @T @T @BASIC 0 @F
@F @F
@T
@BEG_Attrib
3 @RT(0) @RT(0) @RT(0)
@END_Attrib
1 0 @F @F @F @F

@Var @RT(8)TaskSlow @RT(0) @T @F @DT @RT(4)TASK @RT(0) @T @T @BASIC 0 @F
@F @F
@T
@BEG_Attrib
3 @RT(0) @RT(0) @RT(0)
@END_Attrib
1 7 @F @F @F @F

@Var @RT(18)mrTemperatureLimit @RT(0) @T @F @DT @RT(4)REAL @RT(0) @T @T @BASIC 0 @F
@F @F
@T
@BEG_Attrib
3 @RT(0) @RT(0) @RT(0)
@END_Attrib
1 0 @F @F @F @F

@Var @RT(13)erCPUTempHigh @RT(0) @T @F @DT @RT(5)ALARM @RT(0) @T @T @BASIC 0 @F
@F @F
@T
@BEG_Attrib
3 @RT(0) @RT(0) @RT(0)
@END_Attrib
1 7 @F @F @F @F

@END_Dcl

@END_Export

@BEG_Body

4

@BEG_Export

@BEG_Algo
@ALGORITHM @RT(6)aStart @STRUCTURED_TEXT
@RT(0) @RT(0) @RT(0) @F @F
@END_Algo

@BEG_Dcl
@RT(16)DclTreeContainer
0
@END_Dcl

@END_Export

@BEG_Export

@BEG_Algo
@ALGORITHM @RT(5)aStop @STRUCTURED_TEXT
@RT(0) @RT(0) @RT(0) @F @F
@END_Algo

@BEG_Dcl
@RT(16)DclTreeContainer
0
@END_Dcl

@END_Export

@BEG_Export

@BEG_Algo
@PROCESS_ALGORITHM @RT(6)paInit @STRUCTURED_TEXT
@RT(0) @RT(0) @RT(8)TaskSlow @T @F
@END_Algo

@BEG_Dcl
@RT(16)DclTreeContainer
4
@Var @RT(3)hdl @RT(0) @T @T @DERIVED 0 @F @RT(15)KCAT_HandleData @F
@T
@BEG_Attrib
3 @RT(0) @RT(0) @RT(0)
@END_Attrib
1 0 @F @F @F @F

@Var @RT(9)sPlatform @RT(0) @T @F @DT @RT(10)STRING(10) @RT(0) @T @T @STRING 0 @F @RT(2)10 @F
@F @F
@T
@BEG_Attrib
3 @RT(0) @RT(0) @RT(0)
@END_Attrib
1 0 @F @F @F @F

@Var @RT(5)state @RT(0) @T @T @DERIVED 0 @F @RT(11)KCAT_Status @F
@T
@BEG_Attrib
3 @RT(0) @RT(0) @RT(0)
@END_Attrib
1 0 @F @F @F @F

@Var @RT(5)dummy @RT(0) @T @F @DT @RT(4)DINT @RT(0) @T @T @BASIC 0 @F
@F @F
@T
@BEG_Attrib
3 @RT(0) @RT(0) @RT(0)
@END_Attrib
1 0 @F @F @F @F

@END_Dcl

@END_Export

@BEG_Export

@BEG_Algo
@PROCESS_ALGORITHM @RT(5)paRun @STRUCTURED_TEXT
@RT(0) @RT(0) @RT(8)TaskSlow @F @F
@END_Algo

@BEG_Dcl
@RT(16)DclTreeContainer
4
@Var @RT(6)TempID @RT(0) @T @T @DERIVED 0 @T @T @DT @RT(11)KSYS_TempId @RT(0) @T @T @UNKNOWN 0 @F
@F @F
@T
@BEG_Attrib
3 @RT(15)KSYS_TempID_MAB @RT(0) @RT(0)
@END_Attrib
1 0 @F @F @F @F

@Var @RT(8)TempData @RT(0) @T @T @DERIVED 0 @T @T @DT @RT(17)KSYS_GetTemp_Data @RT(0) @T @T @UNKNOWN 0 @F
@F @F
@T
@BEG_Attrib
3 @RT(0) @RT(0) @RT(0)
@END_Attrib
1 0 @F @F @F @F

@Var @RT(9)iCycleRed @RT(0) @T @F @DT @RT(4)DINT @RT(0) @T @T @BASIC 0 @F
@F @F
@T
@BEG_Attrib
3 @RT(0) @RT(0) @RT(0)
@END_Attrib
1 0 @F @F @F @F

@Var @RT(9)bAlarmSet @RT(0) @T @F @DT @RT(4)BOOL @RT(0) @T @T @BASIC 0 @F
@F @F
@T
@BEG_Attrib
3 @RT(0) @RT(0) @RT(0)
@END_Attrib
1 0 @F @F @F @F

@END_Dcl

@END_Export

@BEG_Body
@TL(8)
(**************************************** WARNING ********************************************
 *** The KEBA Kemro K2 System including software is not intended for safety control tasks! ***
 ***                       For further information see Comment tab!                        ***
 *********************************************************************************************)

mbStart := TRUE;
START_PROCESS_ALGORITHM(paRun)

@END_Body

@@@BEG_Comment@@@
@TL(0)

@@@END_Comment@@@

@BEG_Body
@TL(8)
(**************************************** WARNING ********************************************
 *** The KEBA Kemro K2 System including software is not intended for safety control tasks! ***
 ***                       For further information see Comment tab!                        ***
 *********************************************************************************************)

mbStart := FALSE;

@END_Body

@@@BEG_Comment@@@
@TL(0)

@@@END_Comment@@@

@BEG_Body
@TL(24)
(**************************************** WARNING ********************************************
 *** The KEBA Kemro K2 System including software is not intended for safety control tasks! ***
 ***                       For further information see Comment tab!                        ***
 *********************************************************************************************)

//get hardware platform
hdl := KCAT_GetHandle('IRT.Platform');
IF hdl.Status = KCAT_Status_OK THEN
   state := KCAT_GetValue(Handle := hdl.Handle, Buffer := sPlatform);
END_IF;

IF sPlatform = 'PPC' THEN
   mrTemperatureLimit := 83.0; //PPC
ELSIF sPlatform = 'x86' THEN
   mrTemperatureLimit := 115.0; //Intel
ELSE
   //unknown platform -> set trace and use lower temperature limit
   dummy := Print('!!! ABCPUTemperature - paInit: could not detect hardware platform !!!');
   mrTemperatureLimit := 83.0;
END_IF;

mbInit := TRUE;
STOP_PROCESS_ALGORITHM();

@END_Body

@@@BEG_Comment@@@
@TL(0)

@@@END_Comment@@@

@BEG_Body
@TL(34)
(**************************************** WARNING ********************************************
 *** The KEBA Kemro K2 System including software is not intended for safety control tasks! ***
 ***                       For further information see Comment tab!                        ***
 *********************************************************************************************)
IF (NOT mbStart) THEN
    iCycleRed := 0;
    STOP_PROCESS_ALGORITHM();
    RETURN;
END_IF;

IF (NOT mbInit) THEN
    RETURN;
END_IF;

IF ((iCycleRed MOD 64) = 0) THEN // about every 0,5 min
  TempData := GET_TEMP(TempID);

  IF (TempData.Temp >= REAL_TO_DINT(mrTemperatureLimit)) THEN
        SET_ALARM(Name := erCPUTempHigh, Param1 := DINT_TO_STRING(TempData.Temp));
        bAlarmSet := TRUE;
  END_IF;

  IF (TempData.Temp < (REAL_TO_DINT(mrTemperatureLimit) - 1)) THEN
        IF bAlarmSet THEN
            RESET_ALARM(Name := erCPUTempHigh);
            bAlarmSet := FALSE;
        END_IF;
  END_IF;

END_IF;

iCycleRed := iCycleRed + 1;

@END_Body

@@@BEG_Comment@@@
@TL(0)

@@@END_Comment@@@
@END_Body

@END_Contents

(* ---- ABWatchDog.pu ---- *)
IMPORT_OVER_LISTFILE
 GET_WATCHDOG_TERMINAL
, CLOSE_WATCHDOG_TERMINAL
, OPEN_WATCHDOG_TERMINAL
, IS_LINKED
, FREEZE_IOSYSTEM
, SET_ALARM
, RESET_ALARM
, SAVE_TRACE_BUFFER
, SET_TRACE_EVENT_MASK
, WRITE_STAREP
, FGetCatConfigValueString
, GET_STAREP_STATUS
, STOP_PROCESS_ALGORITHM
, START_PROCESS_ALGORITHM
, tsTraceLevel
, KCAT_HandleData
, KSYS_TraceStatus
, KSYS_SysTraceHandleData
, KSYS_Status

END_IMPORT

ALGORITHM_BLOCK ABWatchDog #DUMMY_EDIT_BLOCK

SYSTEM_VAR
 do_Watchdog : BOOL;
 sv_TraceLevel : tsTraceLevel;
END_VAR

SYSTEM_OBJECT
 erWatchdog : ALARM;
 erStarepWriting : ALARM;
 erStarepFinished : ALARM;
 TaskVisLow : TASK;
END_OBJECT

VAR_EXTERNAL
 g_bLinux : BOOL;
END_VAR

VAR
 m_bIOSysFrozen : BOOL := TRUE;
 mbStarepActive : BOOL;
 miStarepState : DINT;
END_VAR

ALGORITHM aSaveTraceBuffer

VAR
 CatHandleUosSystem : KCAT_HandleData;
 CatHandleIecRt : KCAT_HandleData;
 sKpmFileUosSystem : STRING(255) := '/protocol/log/Trace_UOS-System.kpm';
 sKpmFileIecRt : STRING(255) := '/protocol/log/Trace_IecRt.kpm';
 TraceStatus : KSYS_TraceStatus;
 iActUosSystemTraceMask : DWORD;
 iActIecRtTraceMask : DWORD;
 sWorkPath : STRING(255);
 sFTraceFile : STRING(255);
 FTraceHandle : KSYS_SysTraceHandleData (* handle to FTrace *);
END_VAR
#BEGIN_EDIT_BLOCK
(**************************************** WARNING ********************************************
 *** The KEBA Kemro K2 System including software is not intended for safety control tasks! ***
 ***                       For further information see Comment tab!                        ***
 *********************************************************************************************)

CatHandleUosSystem := KCAT_GetHandle('UOS.TRACE.UOS-System-Trace');
IF g_bLinux THEN
   CatHandleIecRt := KCAT_GetHandle('UOS.TRACE.IecRt-CycleTrace0');
ELSE
   CatHandleIecRt := KCAT_GetHandle('UOS.TRACE.IecRt-Trace');
END_IF;

// set event trace masks to 0
iActUosSystemTraceMask := 0;
IF (CatHandleUosSystem.Status = KCAT_Status_OK) THEN
   TraceStatus := GET_TRACE_EVENT_MASK(CatHandleUosSystem.Handle, iActUosSystemTraceMask);
   IF ((TraceStatus = KSYS_TraceStatus_OK) AND (iActUosSystemTraceMask > 0)) THEN
       TraceStatus := SET_TRACE_EVENT_MASK(CatHandleUosSystem.Handle, 0);
   END_IF;
END_IF;

iActIecRtTraceMask := 0;
IF (CatHandleIecRt.Status = KCAT_Status_OK) THEN
   TraceStatus := GET_TRACE_EVENT_MASK(CatHandleIecRt.Handle, iActIecRtTraceMask);
   IF ((TraceStatus = KSYS_TraceStatus_OK) AND (iActIecRtTraceMask > 0)) THEN
       TraceStatus := SET_TRACE_EVENT_MASK(CatHandleIecRt.Handle, 0);
   END_IF;
END_IF;

IF g_bLinux THEN
   FTraceHandle := GET_SYSTEM_TRACE_HANDLE();
   IF (FTraceHandle.Status = KSYS_Status_OK) THEN
      TraceStatus := SET_TRACE_EVENT_MASK(FTraceHandle.Handle, 0);
   END_IF;
END_IF;

// save tracer buffers
sWorkPath := FGetCatConfigValueString('System.workPath', '/harddisk0/');
sKpmFileUosSystem := CONCAT(sWorkPath, sKpmFileUosSystem);
sKpmFileIecRt := CONCAT(sWorkPath, sKpmFileIecRt);

IF g_bLinux THEN
   //save FTrace on linux systems
   sFTraceFile := CONCAT(sWorkPath, '/protocol/log/ftrace.kpm');
   TraceStatus := SAVE_FTRACE_COMPRESSED(TRUE, sFTraceFile);
END_IF;

IF (iActUosSystemTraceMask > 0) THEN
   TraceStatus := SAVE_TRACE_BUFFER(CatHandleUosSystem.Handle, TRUE, sKpmFileUosSystem);
END_IF;

IF (iActIecRtTraceMask > 0) THEN
   TraceStatus := SAVE_TRACE_BUFFER(CatHandleIecRt.Handle, TRUE, sKpmFileIecRt);
END_IF;

;#END_EDIT_BLOCK END_ALGORITHM

ALGORITHM aWriteStarep

VAR
 dummy : DINT;
END_VAR
#BEGIN_EDIT_BLOCK
(**************************************** WARNING ********************************************
 *** The KEBA Kemro K2 System including software is not intended for safety control tasks! ***
 ***                       For further information see Comment tab!                        ***
 *********************************************************************************************)

IF NOT mbStarepActive THEN
    mbStarepActive := TRUE;
    START_PROCESS_ALGORITHM(paCheckStarep);
ELSE
    IF sv_TraceLevel.bExceptionInterpretation THEN
      dummy := Print('ABWatchdog: starep already active - skipping');
    END_IF;
END_IF;

;#END_EDIT_BLOCK END_ALGORITHM

ALGORITHM aOpen

#BEGIN_EDIT_BLOCK
(**************************************** WARNING ********************************************
 *** The KEBA Kemro K2 System including software is not intended for safety control tasks! ***
 ***                       For further information see Comment tab!                        ***
 *********************************************************************************************)

// disable all outputs
FREEZE_IOSYSTEM(Action := TRUE);
m_bIOSysFrozen := TRUE;

IF IS_LINKED(do_Watchdog) THEN
    // external Watchdog Output used
    do_Watchdog := FALSE;
END_IF;

SET_ALARM(Name := erWatchdog);
aSaveTraceBuffer();
aWriteStarep();

;#END_EDIT_BLOCK END_ALGORITHM

ALGORITHM aClose

#BEGIN_EDIT_BLOCK
(**************************************** WARNING ********************************************
 *** The KEBA Kemro K2 System including software is not intended for safety control tasks! ***
 ***                       For further information see Comment tab!                        ***
 *********************************************************************************************)

// allow outputs
FREEZE_IOSYSTEM(Action := FALSE);

IF IS_LINKED(do_Watchdog) THEN
    // external Watchdog Output used
    do_Watchdog := TRUE;
END_IF;

IF m_bIOSysFrozen THEN
    RESET_ALARM(Name := erWatchdog);
END_IF;

m_bIOSysFrozen := FALSE;

;#END_EDIT_BLOCK END_ALGORITHM

ALGORITHM aGet

VAR_OUTPUT
 bState : BOOL;
END_VAR
#BEGIN_EDIT_BLOCK
(**************************************** WARNING ********************************************
 *** The KEBA Kemro K2 System including software is not intended for safety control tasks! ***
 ***                       For further information see Comment tab!                        ***
 *********************************************************************************************)

// getting Watchdog State

IF IS_LINKED(do_Watchdog) THEN
    // external Watchdog Output used
    bState := do_Watchdog;
ELSE
    // no Watchdog Output used
    bState := NOT m_bIOSysFrozen;
END_IF;

;#END_EDIT_BLOCK END_ALGORITHM

PROCESS_ALGORITHM paCheckStarep ON TaskVisLow

VAR
 status : KSYS_Status;
 progress : DWORD;
 starepStatus : DWORD;
 cnt : INT;
 dummy : DINT;
END_VAR
#BEGIN_EDIT_BLOCK
(**************************************** WARNING ********************************************
 *** The KEBA Kemro K2 System including software is not intended for safety control tasks! ***
 ***                       For further information see Comment tab!                        ***
 *********************************************************************************************)

CASE miStarepState OF

    0:  // initiate writing of starep
        status := WRITE_STAREP(); // potentially blocking on Linux

        IF (status = KSYS_Status_OK) THEN
            SET_ALARM(Name := erStarepWriting);
            miStarepState := 1;
        ELSE
            IF sv_TraceLevel.bExceptionInterpretation THEN
                dummy := Print('ABWatchdog: WRITE_STAREP failed - exiting');
            END_IF;
            mbStarepActive := FALSE;
            STOP_PROCESS_ALGORITHM();
        END_IF;

    1: // check starep writing status
        cnt := cnt + 1;
        IF cnt = 10 THEN
            cnt := 0;
        ELSE
            RETURN;
        END_IF;

        status := GET_STAREP_STATUS(starepStatus, progress);
        IF (status = KSYS_Status_OK) THEN
            IF (starepStatus = 0) THEN
                // finished
                RESET_ALARM(Name := erStarepWriting);
                SET_ALARM(Name := erStarepFinished);
                mbStarepActive := FALSE;
                miStarepState := 0;
                STOP_PROCESS_ALGORITHM();
            END_IF;
        ELSE
            // error
            IF sv_TraceLevel.bExceptionInterpretation THEN
                dummy := Print('ABWatchdog: GET_STAREP_STATUS failed - exiting');
            END_IF;
            mbStarepActive := FALSE;
            miStarepState := 0;
            STOP_PROCESS_ALGORITHM();
        END_IF;
ELSE
    IF sv_TraceLevel.bExceptionInterpretation THEN
        dummy := Print('ABWatchdog: invalid starep state machine state %d - exiting', miStarepState);
    END_IF;
    mbStarepActive := FALSE;
    miStarepState := 0;
    STOP_PROCESS_ALGORITHM();
END_CASE;

;#END_EDIT_BLOCK END_ALGORITHM

END_ALGORITHM_BLOCK

#END_OF_IEC_PART

@Puma @IecEditor 6 68 @Pou 25
@@@BEG_Comment@@@

@@@END_Comment@@@

@BEG_Contents

@BEG_Func
@RT(17)FuncTreeContainer
14
@Var @RT(21)GET_WATCHDOG_TERMINAL @RT(0) @T @T @DERIVED 0 @F @RT(22)KEBA_STANDARD_FUNCTION @F
@T
@BEG_Attrib
0 @RT(0) @RT(0)
@END_Attrib
1 1 @F @F @F @F

@Var @RT(23)CLOSE_WATCHDOG_TERMINAL @RT(0) @T @T @DERIVED 0 @F @RT(23)KEBA_STANDARD_PROCEDURE @F
@T
@BEG_Attrib
0 @RT(0) @RT(0)
@END_Attrib
1 1 @F @F @F @F

@Var @RT(22)OPEN_WATCHDOG_TERMINAL @RT(0) @T @T @DERIVED 0 @F @RT(23)KEBA_STANDARD_PROCEDURE @F
@T
@BEG_Attrib
0 @RT(0) @RT(0)
@END_Attrib
1 1 @F @F @F @F

@Var @RT(9)IS_LINKED @RT(0) @T @T @DERIVED 0 @F @RT(22)KEBA_STANDARD_FUNCTION @F
@T
@BEG_Attrib
0 @RT(0) @RT(0)
@END_Attrib
1 1 @F @F @F @F

@Var @RT(15)FREEZE_IOSYSTEM @RT(0) @T @T @DERIVED 0 @F @RT(23)KEBA_STANDARD_PROCEDURE @F
@T
@BEG_Attrib
0 @RT(0) @RT(0)
@END_Attrib
1 1 @F @F @F @F

@Var @RT(9)SET_ALARM @RT(0) @T @T @DERIVED 0 @F @RT(23)KEBA_STANDARD_PROCEDURE @F
@T
@BEG_Attrib
0 @RT(0) @RT(0)
@END_Attrib
1 1 @F @F @F @F

@Var @RT(11)RESET_ALARM @RT(0) @T @T @DERIVED 0 @F @RT(23)KEBA_STANDARD_PROCEDURE @F
@T
@BEG_Attrib
0 @RT(0) @RT(0)
@END_Attrib
1 1 @F @F @F @F

@Var @RT(17)SAVE_TRACE_BUFFER @RT(0) @T @T @DERIVED 0 @F @RT(22)KEBA_STANDARD_FUNCTION @F
@T
@BEG_Attrib
0 @RT(0) @RT(0)
@END_Attrib
1 1 @F @F @F @F

@Var @RT(20)SET_TRACE_EVENT_MASK @RT(0) @T @T @DERIVED 0 @F @RT(22)KEBA_STANDARD_FUNCTION @F
@T
@BEG_Attrib
0 @RT(0) @RT(0)
@END_Attrib
1 1 @F @F @F @F

@Var @RT(12)WRITE_STAREP @RT(0) @T @T @DERIVED 0 @F @RT(22)KEBA_STANDARD_FUNCTION @F
@T
@BEG_Attrib
0 @RT(0) @RT(0)
@END_Attrib
1 1 @F @F @F @F

@Var @RT(24)FGetCatConfigValueString @RT(0) @T @T @DERIVED 0 @F @RT(8)FUNCTION @F
@T
@BEG_Attrib
0 @RT(0) @RT(0)
@END_Attrib
1 1 @F @F @F @F

@Var @RT(17)GET_STAREP_STATUS @RT(0) @T @T @DERIVED 0 @F @RT(22)KEBA_STANDARD_FUNCTION @F
@T
@BEG_Attrib
0 @RT(0) @RT(0)
@END_Attrib
1 1 @F @F @F @F

@Var @RT(22)STOP_PROCESS_ALGORITHM @RT(0) @T @T @DERIVED 0 @F @RT(23)KEBA_STANDARD_PROCEDURE @F
@T
@BEG_Attrib
0 @RT(0) @RT(0)
@END_Attrib
1 1 @F @F @F @F

@Var @RT(23)START_PROCESS_ALGORITHM @RT(0) @T @T @DERIVED 0 @F @RT(23)KEBA_STANDARD_PROCEDURE @F
@T
@BEG_Attrib
0 @RT(0) @RT(0)
@END_Attrib
1 1 @F @F @F @F

@END_Func

@BEG_Const
@RT(18)ConstTreeContainer
0
@END_Const

@BEG_Export

@BEG_Kind
@ALGORITHM_BLOCK @RT(10)ABWatchDog @STRUCTURED_TEXT
@RT(0) @RT(0) @RT(0)
@END_Kind

@BEG_Dcl
@RT(16)DclTreeContainer
10
@Var @RT(10)erWatchdog @RT(0) @T @F @DT @RT(5)ALARM @RT(0) @T @T @BASIC 0 @F
@F @F
@T
@BEG_Attrib
3 @RT(0) @RT(0) @RT(0)
@END_Attrib
1 7 @F @F @F @F

@Var @RT(11)do_Watchdog @RT(0) @T @F @DT @RT(4)BOOL @RT(0) @T @T @BASIC 0 @F
@F @F
@T
@BEG_Attrib
3 @RT(0) @RT(0) @RT(0)
@END_Attrib
1 8 @F @F @F @F

@Var @RT(14)m_bIOSysFrozen @RT(0) @T @F @DT @RT(4)BOOL @RT(0) @T @T @BASIC 0 @F
@F @F
@T
@BEG_Attrib
3 @RT(4)TRUE @RT(0) @RT(0)
@END_Attrib
1 0 @F @F @F @F

@Var @RT(15)erStarepWriting @RT(0) @T @F @DT @RT(5)ALARM @RT(0) @T @T @BASIC 0 @F
@F @F
@T
@BEG_Attrib
3 @RT(0) @RT(0) @RT(0)
@END_Attrib
1 7 @F @F @F @F

@Var @RT(16)erStarepFinished @RT(0) @T @F @DT @RT(5)ALARM @RT(0) @T @T @BASIC 0 @F
@F @F
@T
@BEG_Attrib
3 @RT(0) @RT(0) @RT(0)
@END_Attrib
1 7 @F @F @F @F

@Var @RT(10)TaskVisLow @RT(0) @T @T @RENAMED 0 @T @T @DT @RT(4)TASK @RT(0) @T @T @BASIC 0 @F
@F @F
@T
@BEG_Attrib
3 @RT(0) @RT(0) @RT(0)
@END_Attrib
1 7 @F @F @F @F

@Var @RT(13)sv_TraceLevel @RT(0) @T @T @DERIVED 0 @T @T @DT @RT(12)tsTraceLevel @RT(0) @T @T @UNKNOWN 0 @F
@F @F
@T
@BEG_Attrib
3 @RT(0) @RT(0) @RT(0)
@END_Attrib
1 8 @F @F @F @F

@Var @RT(8)g_bLinux @RT(0) @T @F @DT @RT(4)BOOL @RT(0) @T @T @BASIC 0 @F
@F @F
@T
@BEG_Attrib
3 @RT(0) @RT(0) @RT(0)
@END_Attrib
1 6 @F @F @F @F

@Var @RT(14)mbStarepActive @RT(0) @T @F @DT @RT(4)BOOL @RT(0) @T @T @BASIC 0 @F
@F @F
@T
@BEG_Attrib
3 @RT(0) @RT(0) @RT(0)
@END_Attrib
1 0 @F @F @F @F

@Var @RT(13)miStarepState @RT(0) @T @F @DT @RT(4)DINT @RT(0) @T @T @BASIC 0 @F
@F @F
@T
@BEG_Attrib
3 @RT(0) @RT(0) @RT(0)
@END_Attrib
1 0 @F @F @F @F

@END_Dcl

@END_Export

@BEG_Body

6

@BEG_Export

@BEG_Algo
@ALGORITHM @RT(16)aSaveTraceBuffer @STRUCTURED_TEXT
@RT(0) @RT(0) @RT(0) @F @F
@END_Algo

@BEG_Dcl
@RT(16)DclTreeContainer
10
@Var @RT(18)CatHandleUosSystem @RT(0) @T @T @DERIVED 0 @T @T @DT @RT(15)KCAT_HandleData @RT(0) @T @T @UNKNOWN 0 @F
@F @F
@T
@BEG_Attrib
3 @RT(0) @RT(0) @RT(0)
@END_Attrib
1 0 @F @F @F @F

@Var @RT(14)CatHandleIecRt @RT(0) @T @T @DERIVED 0 @F @RT(15)KCAT_HandleData @F
@T
@BEG_Attrib
3 @RT(0) @RT(0) @RT(0)
@END_Attrib
1 0 @F @F @F @F

@Var @RT(17)sKpmFileUosSystem @RT(0) @T @F @DT @RT(11)STRING(255) @RT(0) @T @T @STRING 0 @F @RT(3)255 @F
@F @F
@T
@BEG_Attrib
3 @RT(36)'/protocol/log/Trace_UOS-System.kpm' @RT(0) @RT(0)
@END_Attrib
1 0 @F @F @F @F

@Var @RT(13)sKpmFileIecRt @RT(0) @T @F @DT @RT(11)STRING(255) @RT(0) @T @T @STRING 0 @F @RT(3)255 @F
@F @F
@T
@BEG_Attrib
3 @RT(31)'/protocol/log/Trace_IecRt.kpm' @RT(0) @RT(0)
@END_Attrib
1 0 @F @F @F @F

@Var @RT(11)TraceStatus @RT(0) @T @T @DERIVED 0 @T @T @DT @RT(16)KSYS_TraceStatus @RT(0) @T @T @UNKNOWN 0 @F
@F @F
@T
@BEG_Attrib
3 @RT(0) @RT(0) @RT(0)
@END_Attrib
1 0 @F @F @F @F

@Var @RT(22)iActUosSystemTraceMask @RT(0) @T @F @DT @RT(5)DWORD @RT(0) @T @T @BASIC 0 @F
@F @F
@T
@BEG_Attrib
3 @RT(0) @RT(0) @RT(0)
@END_Attrib
1 0 @F @F @F @F

@Var @RT(18)iActIecRtTraceMask @RT(0) @T @F @DT @RT(5)DWORD @RT(0) @T @T @BASIC 0 @F
@F @F
@T
@BEG_Attrib
3 @RT(0) @RT(0) @RT(0)
@END_Attrib
1 0 @F @F @F @F

@Var @RT(9)sWorkPath @RT(0) @T @F @DT @RT(11)STRING(255) @RT(0) @T @T @STRING 0 @F @RT(3)255 @F
@F @F
@T
@BEG_Attrib
3 @RT(0) @RT(0) @RT(0)
@END_Attrib
1 0 @F @F @F @F

@Var @RT(11)sFTraceFile @RT(0) @T @F @DT @RT(11)STRING(255) @RT(0) @T @T @STRING 0 @F @RT(3)255 @F
@F @F
@T
@BEG_Attrib
3 @RT(0) @RT(0) @RT(0)
@END_Attrib
1 0 @F @F @F @F

@Var @RT(12)FTraceHandle @RT(0) @T @T @DERIVED 0 @T @T @DT @RT(23)KSYS_SysTraceHandleData @RT(0) @T @T @UNKNOWN 0 @F
@F @F
@T
@BEG_Attrib
3 @RT(0) @RT(16)handle to FTrace @RT(0)
@END_Attrib
1 0 @F @F @F @F

@END_Dcl

@END_Export

@BEG_Export

@BEG_Algo
@ALGORITHM @RT(12)aWriteStarep @STRUCTURED_TEXT
@RT(0) @RT(0) @RT(0) @F @F
@END_Algo

@BEG_Dcl
@RT(16)DclTreeContainer
1
@Var @RT(5)dummy @RT(0) @T @F @DT @RT(4)DINT @RT(0) @T @T @BASIC 0 @F
@F @F
@T
@BEG_Attrib
3 @RT(0) @RT(0) @RT(0)
@END_Attrib
1 0 @F @F @F @F

@END_Dcl

@END_Export

@BEG_Export

@BEG_Algo
@ALGORITHM @RT(5)aOpen @STRUCTURED_TEXT
@RT(0) @RT(0) @RT(0) @F @F
@END_Algo

@BEG_Dcl
@RT(16)DclTreeContainer
0
@END_Dcl

@END_Export

@BEG_Export

@BEG_Algo
@ALGORITHM @RT(6)aClose @STRUCTURED_TEXT
@RT(0) @RT(0) @RT(0) @F @F
@END_Algo

@BEG_Dcl
@RT(16)DclTreeContainer
0
@END_Dcl

@END_Export

@BEG_Export

@BEG_Algo
@ALGORITHM @RT(4)aGet @STRUCTURED_TEXT
@RT(6)bState @RT(0) @RT(0) @F @F
@END_Algo

@BEG_Dcl
@RT(16)DclTreeContainer
1
@Var @RT(6)bState @RT(0) @T @F @DT @RT(4)BOOL @RT(0) @T @T @BASIC 0 @F
@F @F
@T
@BEG_Attrib
3 @RT(0) @RT(0) @RT(0)
@END_Attrib
1 3 @F @F @F @F

@END_Dcl

@END_Export

@BEG_Export

@BEG_Algo
@PROCESS_ALGORITHM @RT(13)paCheckStarep @STRUCTURED_TEXT
@RT(0) @RT(0) @RT(10)TaskVisLow @F @F
@END_Algo

@BEG_Dcl
@RT(16)DclTreeContainer
5
@Var @RT(6)status @RT(0) @T @T @DERIVED 0 @T @T @DT @RT(11)KSYS_Status @RT(0) @T @T @UNKNOWN 0 @F
@F @F
@T
@BEG_Attrib
3 @RT(0) @RT(0) @RT(0)
@END_Attrib
1 0 @F @F @F @F

@Var @RT(8)progress @RT(0) @T @F @DT @RT(5)DWORD @RT(0) @T @T @BASIC 0 @F
@F @F
@T
@BEG_Attrib
3 @RT(0) @RT(0) @RT(0)
@END_Attrib
1 0 @F @F @F @F

@Var @RT(12)starepStatus @RT(0) @T @F @DT @RT(5)DWORD @RT(0) @T @T @BASIC 0 @F
@F @F
@T
@BEG_Attrib
3 @RT(0) @RT(0) @RT(0)
@END_Attrib
1 0 @F @F @F @F

@Var @RT(3)cnt @RT(0) @T @F @DT @RT(3)INT @RT(0) @T @T @BASIC 0 @F
@F @F
@T
@BEG_Attrib
3 @RT(0) @RT(0) @RT(0)
@END_Attrib
1 0 @F @F @F @F

@Var @RT(5)dummy @RT(0) @T @F @DT @RT(4)DINT @RT(0) @T @T @BASIC 0 @F
@F @F
@T
@BEG_Attrib
3 @RT(0) @RT(0) @RT(0)
@END_Attrib
1 0 @F @F @F @F

@END_Dcl

@END_Export

@BEG_Body
@TL(58)
(**************************************** WARNING ********************************************
 *** The KEBA Kemro K2 System including software is not intended for safety control tasks! ***
 ***                       For further information see Comment tab!                        ***
 *********************************************************************************************)

CatHandleUosSystem := KCAT_GetHandle('UOS.TRACE.UOS-System-Trace');
IF g_bLinux THEN
   CatHandleIecRt := KCAT_GetHandle('UOS.TRACE.IecRt-CycleTrace0');
ELSE
   CatHandleIecRt := KCAT_GetHandle('UOS.TRACE.IecRt-Trace');
END_IF;

// set event trace masks to 0
iActUosSystemTraceMask := 0;
IF (CatHandleUosSystem.Status = KCAT_Status_OK) THEN
   TraceStatus := GET_TRACE_EVENT_MASK(CatHandleUosSystem.Handle, iActUosSystemTraceMask);
   IF ((TraceStatus = KSYS_TraceStatus_OK) AND (iActUosSystemTraceMask > 0)) THEN
       TraceStatus := SET_TRACE_EVENT_MASK(CatHandleUosSystem.Handle, 0);
   END_IF;
END_IF;

iActIecRtTraceMask := 0;
IF (CatHandleIecRt.Status = KCAT_Status_OK) THEN
   TraceStatus := GET_TRACE_EVENT_MASK(CatHandleIecRt.Handle, iActIecRtTraceMask);
   IF ((TraceStatus = KSYS_TraceStatus_OK) AND (iActIecRtTraceMask > 0)) THEN
       TraceStatus := SET_TRACE_EVENT_MASK(CatHandleIecRt.Handle, 0);
   END_IF;
END_IF;

IF g_bLinux THEN
   FTraceHandle := GET_SYSTEM_TRACE_HANDLE();
   IF (FTraceHandle.Status = KSYS_Status_OK) THEN
      TraceStatus := SET_TRACE_EVENT_MASK(FTraceHandle.Handle, 0);
   END_IF;
END_IF;

// save tracer buffers
sWorkPath := FGetCatConfigValueString('System.workPath', '/harddisk0/');
sKpmFileUosSystem := CONCAT(sWorkPath, sKpmFileUosSystem);
sKpmFileIecRt := CONCAT(sWorkPath, sKpmFileIecRt);

IF g_bLinux THEN
   //save FTrace on linux systems
   sFTraceFile := CONCAT(sWorkPath, '/protocol/log/ftrace.kpm');
   TraceStatus := SAVE_FTRACE_COMPRESSED(TRUE, sFTraceFile);
END_IF;

IF (iActUosSystemTraceMask > 0) THEN
   TraceStatus := SAVE_TRACE_BUFFER(CatHandleUosSystem.Handle, TRUE, sKpmFileUosSystem);
END_IF;

IF (iActIecRtTraceMask > 0) THEN
   TraceStatus := SAVE_TRACE_BUFFER(CatHandleIecRt.Handle, TRUE, sKpmFileIecRt);
END_IF;

@END_Body

@@@BEG_Comment@@@
@TL(0)

@@@END_Comment@@@

@BEG_Body
@TL(16)
(**************************************** WARNING ********************************************
 *** The KEBA Kemro K2 System including software is not intended for safety control tasks! ***
 ***                       For further information see Comment tab!                        ***
 *********************************************************************************************)

IF NOT mbStarepActive THEN
    mbStarepActive := TRUE;
    START_PROCESS_ALGORITHM(paCheckStarep);
ELSE
    IF sv_TraceLevel.bExceptionInterpretation THEN
      dummy := Print('ABWatchdog: starep already active - skipping');
    END_IF;
END_IF;

@END_Body

@@@BEG_Comment@@@
@TL(0)

@@@END_Comment@@@

@BEG_Body
@TL(18)
(**************************************** WARNING ********************************************
 *** The KEBA Kemro K2 System including software is not intended for safety control tasks! ***
 ***                       For further information see Comment tab!                        ***
 *********************************************************************************************)

// disable all outputs
FREEZE_IOSYSTEM(Action := TRUE);
m_bIOSysFrozen := TRUE;

IF IS_LINKED(do_Watchdog) THEN
    // external Watchdog Output used
    do_Watchdog := FALSE;
END_IF;

SET_ALARM(Name := erWatchdog);
aSaveTraceBuffer();
aWriteStarep();

@END_Body

@@@BEG_Comment@@@
@TL(0)

@@@END_Comment@@@

@BEG_Body
@TL(21)
(**************************************** WARNING ********************************************
 *** The KEBA Kemro K2 System including software is not intended for safety control tasks! ***
 ***                       For further information see Comment tab!                        ***
 *********************************************************************************************)

// allow outputs
FREEZE_IOSYSTEM(Action := FALSE);

IF IS_LINKED(do_Watchdog) THEN
    // external Watchdog Output used
    do_Watchdog := TRUE;
END_IF;

IF m_bIOSysFrozen THEN
    RESET_ALARM(Name := erWatchdog);
END_IF;

m_bIOSysFrozen := FALSE;

@END_Body

@@@BEG_Comment@@@
@TL(0)

@@@END_Comment@@@

@BEG_Body
@TL(16)
(**************************************** WARNING ********************************************
 *** The KEBA Kemro K2 System including software is not intended for safety control tasks! ***
 ***                       For further information see Comment tab!                        ***
 *********************************************************************************************)

// getting Watchdog State

IF IS_LINKED(do_Watchdog) THEN
    // external Watchdog Output used
    bState := do_Watchdog;
ELSE
    // no Watchdog Output used
    bState := NOT m_bIOSysFrozen;
END_IF;

@END_Body

@@@BEG_Comment@@@
@TL(0)

@@@END_Comment@@@

@BEG_Body
@TL(62)
(**************************************** WARNING ********************************************
 *** The KEBA Kemro K2 System including software is not intended for safety control tasks! ***
 ***                       For further information see Comment tab!                        ***
 *********************************************************************************************)

CASE miStarepState OF

    0:  // initiate writing of starep
        status := WRITE_STAREP(); // potentially blocking on Linux

        IF (status = KSYS_Status_OK) THEN
            SET_ALARM(Name := erStarepWriting);
            miStarepState := 1;
        ELSE
            IF sv_TraceLevel.bExceptionInterpretation THEN
                dummy := Print('ABWatchdog: WRITE_STAREP failed - exiting');
            END_IF;
            mbStarepActive := FALSE;
            STOP_PROCESS_ALGORITHM();
        END_IF;

    1: // check starep writing status
        cnt := cnt + 1;
        IF cnt = 10 THEN
            cnt := 0;
        ELSE
            RETURN;
        END_IF;

        status := GET_STAREP_STATUS(starepStatus, progress);
        IF (status = KSYS_Status_OK) THEN
            IF (starepStatus = 0) THEN
                // finished
                RESET_ALARM(Name := erStarepWriting);
                SET_ALARM(Name := erStarepFinished);
                mbStarepActive := FALSE;
                miStarepState := 0;
                STOP_PROCESS_ALGORITHM();
            END_IF;
        ELSE
            // error
            IF sv_TraceLevel.bExceptionInterpretation THEN
                dummy := Print('ABWatchdog: GET_STAREP_STATUS failed - exiting');
            END_IF;
            mbStarepActive := FALSE;
            miStarepState := 0;
            STOP_PROCESS_ALGORITHM();
        END_IF;
ELSE
    IF sv_TraceLevel.bExceptionInterpretation THEN
        dummy := Print('ABWatchdog: invalid starep state machine state %d - exiting', miStarepState);
    END_IF;
    mbStarepActive := FALSE;
    miStarepState := 0;
    STOP_PROCESS_ALGORITHM();
END_CASE;

@END_Body

@@@BEG_Comment@@@
@TL(0)

@@@END_Comment@@@
@END_Body

@END_Contents
